FUNCTION_BLOCK F_MID (* L characters of IN *)
  PACKAGE iec61131::charString;
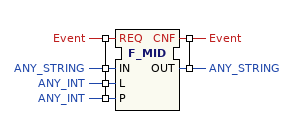
  EVENT_INPUT
    REQ WITH IN, L, P; (* Service Request *)
  END_EVENT
  EVENT_OUTPUT
    CNF WITH OUT; (* Confirmation of Requested Service *)
  END_EVENT
  VAR_INPUT
    IN : ANY_STRING; (* characters *)
    L : ANY_INT; (* length *)
    P : ANY_INT; (* start position *)
  END_VAR
  VAR_OUTPUT
    OUT : ANY_STRING; (* substring from P to P+L *)
  END_VAR
END_FUNCTION_BLOCK
